FUNCTION_BLOCK FB_RCC_TEST EXTENDS FB_TestSuite
VAR_INPUT
END_VAR
VAR_OUTPUT
END_VAR
VAR
END_VAR

END_FUNCTION_BLOCK

(* stored: Version 1.1.0.1, ProductVersion 3.1.4024.12
   POU FB_RCC_TEST: Id {601daf38-e4c9-4c7e-b134-2d83b8bfe7a2}, SpecialFunc None *)
